(* PLC project  *)

CONFIGURATION Empty_Module_17
END_CONFIGURATION
